Staubli VAL3: Save.pgx

program Save()
  local num l_ni
begin
  //
  prd:libSave()
  popUpMsg("保存完毕!")
end
